(* PLC project Generated.project, CODESYS CODESYS V3.5 SP19 Patch 1 *)
(* stored: creationDateTime 2026-11-18T03:01:31.743540, modificationDateTime 2026-11-18T03:01:31.743540 *)

(* ======================================================================= 💾 ST_Encoder_Calib — Calibration & référence codeur (1 par treuil, RETAIN) ─────────────────────────────────────────────────────────────── 🎯 Rôle : Structure de calibration RETAIN par treuil (M1_EncoderCalib / M2_EncoderCalib) 💾 Données : Références brutes, état homed et contrôle de cohérence redémarrage 📄 Doc métier : DOC/AF/AF_Partie-09_Fonction_Encoder_v2.4.md ======================================================================= *)
TYPE ST_Encoder_Calib : STRUCT
  HomingRefRaw : UDINT;  (* === DONNEES DE REFERENCE BRUTE (RETAIN) === Valeur brute figee au dernier homing reussi *)
  LastKnownRawPos : UDINT;  (* Dernier point brut valide connu (continu) *)
  RestartCoherenceTolerancePts : UDINT := 1000;  (* === CONFIGURATION & REGLAGES TOLERANCE === Tolerance redemarrage (pts, ~12% de 8192) *)
  Homed : BOOL;  (* === ETATS DE CALIBRATION & SECURITE === TRUE des qu'un referencement a reussi *)
  HomingSuspect : BOOL;  (* TRUE si incoherence detectee au redemarrage *)
  HomingProvisional : BOOL;  (* TRUE si zero provisoire 0m HX1 (avant HX4 8.5m) *)
END_STRUCT;
END_TYPE

(* ======================================================================= 🧩 ST_Fault — Brique socle défaut (2 vues : live + latchée) ─────────────────────────────────────────────────────────────── 🎯 Rôle : porter l'état défaut d'un composant, applicable dans TOUS les cas (acquittable ou non), sans brique warning séparée. • Vue LIVE (Error / ErrorId) : suit la cause, retombe seule à 0. • Vue LATCHÉE (Latched / LatchedId): mémorisée au défaut, reste jusqu'au front Reset. Le choix acquittable / non-acquittable se fait PAR CAUSE (ST_FaultCause.Latching), jamais par bloc. 🔒 Sécurité : interlock TOUJOURS sur la cause brute (Error / ErrorId), jamais sur l'acquittement. Reset TOUJOURS effectif, jamais conditionné (std §9). 🧬 Composition : brique de base réutilisable — sortie de FB, struct métier, GVL. Texte IHM NON stocké ici : dérivé côté IHM depuis LatchedId / ErrorId. 📄 Doc : DOC/STDS/CODE_QUALITY_STANDARDS.md §2quinquies / §9 ======================================================================= *)
TYPE ST_Fault : STRUCT
  Error : BOOL;  (* <-- [DIAG] vue LIVE : au moins une cause présente maintenant *)
  ErrorId : WORD;  (* <-- [DIAG] bitfield des causes présentes maintenant (0 si aucune) *)
  Latched : BOOL;  (* <-- [DIAG] vue LATCHÉE : défaut non acquitté, reste jusqu'au front Reset *)
  LatchedId : WORD;  (* <-- [DIAG] ErrorId figé à l'apparition du défaut, effacé au Reset *)
END_STRUCT;
END_TYPE

(* ======================================================================= 🧩 ST_FaultCause — Cause élémentaire alimentant ST_Fault (socle FB_FaultCore) ─────────────────────────────────────────────────────────────── 🎯 Rôle : une cause exprimée EN CLAIR (BOOL + libellé), sans bitfield ni masque. Le FB métier remplit une liste (ARRAY[0..15] OF ST_FaultCause) ; le socle FB_FaultCore en déduit ST_Fault (vue live + vue latchée). 🔒 Sécurité : interlock TOUJOURS sur Active (cause brute), jamais sur le latch. Latching = TRUE → la cause ARME la vue latchée (défaut à acquitter). Latching = FALSE → la cause n'alimente que la vue live (retombe seule). Fail-safe : une cause laissée à Latching=FALSE reste visible en live — pour la rendre acquittable, il faut le déclarer explicitement. 📄 Doc : DOC/STDS/CODE_QUALITY_STANDARDS.md §2quinquies / §9 ======================================================================= *)
TYPE ST_FaultCause : STRUCT
  Active : BOOL;  (* 1 = cause présente maintenant (interlock sur cette valeur) *)
  Latching : BOOL;  (* 1 = cause à acquitter (arme Latched) ; 0 = live seulement *)
  Texte : STRING;  (* libellé prêt IHM (non stocké dans ST_Fault, dérivé côté IHM) *)
END_STRUCT;
END_TYPE

(* ======================================================================= ⚙️ ST_fbEncoder_Cfg — Réglages technologiques publics de FB_Encoder ─────────────────────────────────────────────────────────────────────── 🎯 Rôle : porter le mode de confirmation preset commun aux codeurs. 🔒 Ownership : GVL_IHM.Commun.EncoderCfg ↔ GVL_PERSISTENT._EncoderCfgPersist. 📄 Doc : DOC/AF/AF_Partie-09_Fonction_Encoder_v2.4.md ======================================================================= *)
TYPE ST_fbEncoder_Cfg : STRUCT
  PresetConfirmMode : E_PresetConfirmMode := E_PresetConfirmMode.READBACK_ONLY;  (* Mode de confirmation preset, défaut relecture *)
  Initialized : BOOL := FALSE;  (* 🚦 TRUE après restauration du pont persistant *)
END_STRUCT;
END_TYPE

(* ======================================================================= 🔌 ST_fbEncoder_HwIn — Faits hardware d'entrée codeur (HwIn) ─────────────────────────────────────────────────────────────── 🎯 Rôle : Regrouper les SEULES entrées/faits hardware d'un codeur absolu EtherCAT consommés par FB_Encoder (lecture seule côté automate). 🔒 Ownership : PRG_02_Acquisition câble ce bus depuis le device/simulé. 🛡️ PresetStatusBit : bit du mot d'état codeur, réservé site futur — câblé à FALSE tant qu'aucun bit n'est identifié (aucun signal absent ne confirme implicitement le preset). 📄 Doc métier : DOC/AF/AF_Partie-09_Fonction_Encoder_v2.4.md ======================================================================= *)
TYPE ST_fbEncoder_HwIn : STRUCT
  RawPosIn : UDINT;  (* === ENTRÉES BUS ETHERCAT (faits d'entrée, lecture seule) === --> [HW] Position brute codeur *)
  SpdValueIn : DINT;  (* --> [HW] Vitesse brute codeur (0x6031:01 en 0.1 RPM) *)
  AlarmsIn : UINT;  (* --> [HW] Alarmes brutes codeur *)
  WarningsIn : UINT;  (* --> [HW] Avertissements bruts codeur *)
  SlaveOperational : BOOL;  (* --> [HW] Esclave EtherCAT operationnel *)
  PresetStatusBit : BOOL;  (* --> [HW] Bit d'etat preset optionnel, FALSE si non cable *)
END_STRUCT;
END_TYPE

(* ======================================================================= 🔌 ST_fbEncoder_HwOut — Ordres preset de sortie codeur (HwOut) ─────────────────────────────────────────────────────────────── 🎯 Rôle : Regrouper les SEULES sorties/ordres preset d'un codeur absolu EtherCAT produits par FB_Encoder vers le PDO Rx (bus sortie). 🔒 Ownership : FB_Encoder produit ce bus ; PRG_02_Acquisition le relaie vers le device. 📄 Doc métier : DOC/AF/AF_Partie-09_Fonction_Encoder_v2.4.md ======================================================================= *)
TYPE ST_fbEncoder_HwOut : STRUCT
  PresetTriggerCmd : WORD;  (* === SORTIES BUS ETHERCAT (ordres preset vers PDO Rx) === <-- [ACT] Declenchement preset vers PDO Rx *)
  CodeSeqTriggerCmd : WORD;  (* <-- [ACT] Sequence code vers PDO Rx, maintenue a 0 *)
  PresetValueOut : UDINT;  (* <-- [ACT] Valeur brute envoyee au preset *)
END_STRUCT;
END_TYPE

(* ======================================================================= 📊 ST_fbEncoder_Measurement — Mesures codeur conditionnées (1 sous-DUT par treuil) ─────────────────────────────────────────────────────────────── 🎯 Rôle : Regroupement des mesures et faits de la chaîne codeur d'un treuil (Abs → Scale → Safety → Speed) 🔌 Interface : Interface de mesure normalisée pour PRG_02_Acquisition 📄 Doc métier : DOC/AF/AF_Partie-06_Acquisition_Qualification_IO_v2.4.md ======================================================================= *)
TYPE ST_fbEncoder_Measurement : STRUCT
  RawPos : UDINT;  (* === DONNEES BRUTES & STATUT BUS === Position brute codeur (gelee si EncoderAvailable=FALSE) *)
  EncoderAvailable : BOOL;  (* TRUE = bus/esclave EtherCAT operationnel et disponible *)
  CablePosM : REAL;  (* === MESURES DE POSITION CABLE === Position cable (m, signee, + enroule) *)
  CablePosMSafe : REAL;  (* Position cable instantanee validee par EncoderIncoherent (m) *)
  EncoderIncoherent : BOOL;  (* TRUE = incoherence redemarrage ou hors bornes *)
  Speed_Mps : REAL;  (* === MESURES DE VITESSE CABLE === Vitesse absolue câble (m/s) *)
  SignedSpeed_Mps : REAL;  (* Vitesse signee câble (m/s, + montee, - descente) *)
  SpeedValid : BOOL;  (* TRUE si mesure valide et codeur operationnel *)
  HomingFault : ST_Fault;  (* === STATUTS DES SOUS-FB & REFERENCE === Défaut FB_Encoder_Homing (état du référencement) *)
  HomingLifecycle : ST_Lifecycle;  (* Cycle FB_Encoder_Homing (Busy/Done) *)
  AbsFault : ST_Fault;  (* Défaut FB_Encoder_Abs (état acquisition bus) *)
  HomingRefRaw : UDINT;  (* Reference brute du dernier homing reussi (re-expose) *)
END_STRUCT;
END_TYPE

(* ======================================================================= 🧩 ST_Lifecycle — Brique socle cycle d'exécution ─────────────────────────────────────────────────────────────── 🎯 Rôle : porter l'avancement d'une action à cycle (organe, séquenceur). Optionnelle : un FB purement synchrone (conditionneur, filtre, joystick) ne la porte pas. 🧬 Composition : brique de base réutilisable, composée avec ST_Fault. 📄 Doc : DOC/STDS/CODE_QUALITY_STANDARDS.md §2quinquies ======================================================================= *)
TYPE ST_Lifecycle : STRUCT
  Busy : BOOL;  (* <-- [STAT] 1 = action en cours *)
  Done : BOOL;  (* <-- [STAT] 1 = action terminée avec succès *)
END_STRUCT;
END_TYPE

(* values of E_PresetConfirmMode: READBACK_ONLY: Confirmation par relecture de position; READBACK_AND_STATUSBIT: Relecture et bit d'état matériel; STATUSBIT_ONLY: Bit d'état matériel uniquement *)

{attribute 'qualified_only'}
{attribute 'strict'}
TYPE E_PresetConfirmMode : (READBACK_ONLY := 0, READBACK_AND_STATUSBIT := 1, STATUSBIT_ONLY := 2);
END_TYPE

(* ======================================================================= 🔌 FB_Encoder — Objet codeur complet (1 par treuil M1/M2) ─────────────────────────────────────────────────────────────── 🎯 Rôle : Regrouper toute la chaine codeur derriere une interface unique : Abs → Homing → Scale → Safety → Reliability → Speed. 🔌 Frontiere hardware separee HwIn/HwOut (testable). 🔒 Homing : autorise par HomingPermit (calcule par le caller), declenche par HomingAtTargetM (front). La cible est fournie par le caller. 🔒 Fiabilite : gate EncoderFault (sans Homed) calcule AVANT Speed — purge de vitesse au meme scan. HomedAndReliable = gate strict interlock M3. 🧩 Defaut : Fault:ST_Fault rempli par FB_FaultCore (instFault) depuis une liste de causes en clair (instCauses) — pattern FB_Joystick. Ready = Enable ET pas de defaut late. Interlocks machine sur les faits bruts, jamais sur Fault.Latched. 📄 Doc : DOC/AF/AF_Partie-09_Fonction_Encoder_v2.4.md ======================================================================= *)
FUNCTION_BLOCK FB_Encoder
  VAR_INPUT
    Enable : BOOL;  (* === COMMANDES & AUTORISATIONS === --> [CMD] Autorisation generale FB (TRUE=Autorise) *)
    Reset : BOOL;  (* --> [CMD] Acquittement defaut (front montant) *)
    HomingPermit : BOOL;  (* === AUTORISATION HOMING (calculee par le caller PRG) === --> [CMD] TRUE = l'operateur a le droit de homer *)
    HomingAtTargetM : BOOL;  (* === CONSIGNES HOMING === --> [CMD] Demande homing vers cible (front montant) *)
    HomingAtZero : BOOL;  (* --> [CMD] Force homing a 0.0 *)
    ConfirmCoherence : BOOL;  (* --> [CMD] Lever le doute d'incoherence boot *)
    CfgHomingTargetM : REAL;  (* --> [CFG] Cible libre homing unitaire (m) *)
    CfgTopSensorPosM : REAL;  (* --> [CFG] Cible homing nominal capteur haut (m) *)
    UseDynamicTarget : BOOL;  (* --> [CMD] Active cible dynamique *)
    DynamicHomingTargetM : REAL;  (* --> [CFG] Cible dynamique de referencement (m) *)
    InvalidateDatum : BOOL := FALSE;  (* --> [CMD] Invalidation explicite du datum (abandon homing avant altimetrie) *)
    ProvisionalHoming : BOOL := FALSE;  (* --> [CMD] TRUE = zero provisoire HX1 (survive coupure secteur RETAIN) *)
    TopPositionSensor : BOOL;  (* === CAPTEURS PHYSIQUES === --> [HW] Capteur physique position haute unique *)
    HwIn : ST_fbEncoder_HwIn;  (* === BUS ETHERCAT & CAPTEUR HW (frontiere testable) === --> [HW] Retours hardware codeur *)
    PointsPerRev : UDINT := 8192;  (* === MECANIQUE (constantes) === --> [CFG] Resolution codeur (pts/tour) *)
    CableM_PerRev : REAL := 2;  (* --> [CFG] Developpement cable par tour (m/tour) *)
    Cfg : ST_fbEncoder_Cfg;  (* === REGLAGES & CONFIGURATION === --> [CFG] Mode de confirmation preset *)
    PositionMinM : REAL := -99;  (* --> [CFG] Plafond bornage physique bas (m) *)
    PositionMaxM : REAL := 99;  (* --> [CFG] Plafond bornage physique haut (m) *)
    BypassGlobal : BOOL := FALSE;  (* --> [TST] Neutralisation defauts pour mise en service *)
  END_VAR
  VAR_OUTPUT
    Ready : BOOL;  (* === ETATS IEC & SYNOPTIQUE === <-- [STAT] FB pret a fonctionner (Enable ET pas de defaut late) *)
    Fault : ST_Fault;  (* <-- [DIAG] Brique defaut socle (live + latchee), remplie par FB_FaultCore *)
    HwOut : ST_fbEncoder_HwOut;  (* === FRONTIERE HW SORTIE (testable) === <-- [ACT] Ordres hardware codeur (preset) *)
    Measurement : ST_fbEncoder_Measurement;  (* === MESURES CONDITIONNEES (struct frontiere) === <-- [BUS] Mesures + statuts (interface) *)
    Homed : BOOL;  (* === ETATS CODEUR === <-- [STAT] Codeur reference (sortie homing) *)
    HomingSuspect : BOOL;  (* <-- [DIAG] Incoherence redemarrage a lever *)
    HomingProvisional : BOOL;  (* <-- [STAT] TRUE si datum provisoire RETAIN actif (HX1 0m) *)
    EncoderFault : BOOL;  (* <-- [SAFE] Gate general fiabilite (sans Homed) *)
    HomedAndReliable : BOOL;  (* <-- [STAT] Gate strict M3 : dispo ET ref ET pas incoherent *)
    PresetConfirmationFailed : BOOL;  (* <-- [DIAG] Latch derniere verification preset echouee *)
  END_VAR
  VAR_IN_OUT
    Calib : ST_Encoder_Calib;  (* === CALIBRATION PERSISTANTE (externe RETAIN, jamais membre) === <-> [BUS] Calibration RETAIN du treuil *)
  END_VAR
  VAR
    instAbs : FB_Encoder_Abs;  (* === SOUS-INSTANCES FB (chaine codeur complete) === * [INST] Acquisition brute codeur EtherCAT *)
    instHoming : FB_Encoder_Homing;  (* * [INST] Referencement (homing) nominal/unitaire *)
    instScale : FB_Encoder_Scale;  (* * [INST] Mise a l'echelle points -> metres *)
    instSafety : FB_Encoder_Safety;  (* * [INST] Bornage & coherence mesure *)
    instRel : FB_EncoderReliability;  (* * [INST] Gates de fiabilite *)
    instSpeed : FB_Encoder_SpeedMeasure;  (* * [INST] Calcul vitesse cable *)
    instFault : FB_FaultCore;  (* * [INST] Socle de defaut (liste de causes -> ST_Fault) *)
    instCauses : ARRAY[0..15] OF ST_FaultCause;  (* . [LOC] Liste des causes pour le socle FB_FaultCore *)
  END_VAR

            

{region "§1 Gate neutralisation"}
IF NOT Enable THEN
    Ready := FALSE;
    Measurement.RawPos := 0; Measurement.EncoderAvailable := FALSE;
    Measurement.CablePosM := 0.0; Measurement.CablePosMSafe := 0.0; Measurement.EncoderIncoherent := FALSE;
    Measurement.Speed_Mps := 0.0; Measurement.SignedSpeed_Mps := 0.0; Measurement.SpeedValid := FALSE;
    Measurement.HomingFault.Error := FALSE; Measurement.HomingFault.ErrorId := 0;
    Measurement.HomingLifecycle.Busy := FALSE; Measurement.HomingLifecycle.Done := FALSE;
    Measurement.AbsFault.Error := FALSE;    Measurement.AbsFault.ErrorId := 0;
    EncoderFault := TRUE;
    HomedAndReliable := FALSE;
    // Frontiere HW sortie : aucun ordre preset publie hors autorisation
    // (sinon PRG_02_Acquisition relaie une valeur perimee au codeur absolu -> preset parasite, reference corrompue)
    HwOut.PresetTriggerCmd := 0; HwOut.CodeSeqTriggerCmd := 0; HwOut.PresetValueOut := 0;
    // Reference connue MAINTENUE depuis Calib (RETAIN) meme FB desactive (AF09 §4) :
    // un FB desactive ne doit pas faire perdre la reference aux consommateurs aval (PRG_04, FB_Encoder_Scale).
    Homed := Calib.Homed;
    HomingSuspect := Calib.HomingSuspect;
    HomingProvisional := Calib.HomingProvisional;
    Measurement.HomingRefRaw := Calib.HomingRefRaw;
    // PresetConfirmationFailed est un diagnostic latch : il reste gele hors Enable
    // et ne doit pas etre efface par ce gate (AC3).
    // Socle appele meme Enable=FALSE : maintient le latch non acquitte et traite le Reset
    // hors autorisation (AC4). Les causes ne sont pas evaluees (Enable=FALSE -> vue live a 0),
    // les latches sont preserves.
    instFault(Enable := FALSE, Reset := Reset, Causes := instCauses);
    Fault := instFault.Fault;
    RETURN;
END_IF;
Ready := TRUE;
{endregion}

{region "§2 Abs"}
    instAbs(
    Enable              := Enable,
    Reset               := Reset,
    RawPosIn            := HwIn.RawPosIn,
    AlarmsIn            := HwIn.AlarmsIn,
    WarningsIn          := HwIn.WarningsIn,
    SlaveOperational    := HwIn.SlaveOperational,
    PresetRequest       := instHoming.PresetRequest,
    PresetValue         := instHoming.PresetValue,
    PointsPerRev        := PointsPerRev
);
{endregion}

{region "§3 Homing"}
instHoming(
    Enable               := Enable,
    Reset                := Reset,
    Home                 := HomingAtTargetM,
    HomingPermit         := HomingPermit,
    BtnConfirmCoherence  := ConfirmCoherence,
    InvalidateDatum      := InvalidateDatum,
    ProvisionalHoming    := ProvisionalHoming,
    UseDynamicTarget     := UseDynamicTarget,
    DynamicHomingTargetM := DynamicHomingTargetM,
    CfgHomingTargetM     := CfgHomingTargetM,
    CfgTopSensorPosM     := SEL(HomingAtZero, CfgTopSensorPosM, 0.0),
    TopPositionSensor    := TopPositionSensor,
    RawPos               := instAbs.RawPos,
    EncoderAvailable     := instAbs.EncoderAvailable,
    PresetStatusBit      := HwIn.PresetStatusBit,
    Cfg                  := Cfg,
    PointsPerRev         := PointsPerRev,
    MultiTurnRevsMax     := 4096,
    CableM_PerRev        := CableM_PerRev,
    BypassGlobal         := BypassGlobal,
    Calib                := Calib
);
{endregion}

{region "§4 Scale"}
instScale(
    RawPos       := instAbs.RawPos,
    HomingRefRaw := instHoming.HomingRefRaw,
    CableM_PerRev := CableM_PerRev,
    PointsPerRev := PointsPerRev
);
{endregion}

{region "§5 Safety"}
instSafety(
    Enable             := Enable,
    Reset              := Reset,
    CablePosM          := instScale.CablePosM,
    HomingSuspect      := instHoming.HomingSuspect,
    PositionMinM       := PositionMinM,
    PositionMaxM       := PositionMaxM,
    BypassGlobal       := BypassGlobal
);
{endregion}

{region "§6 Reliability"}
instRel(
    EncoderAvailable  := instAbs.EncoderAvailable,
    Homed             := instHoming.Homed,
    EncoderIncoherent := instSafety.EncoderIncoherent
);
{endregion}

{region "§7 Speed"}
instSpeed(
    Enable        := Enable,
    Reset         := Reset,
    SpdValueIn    := HwIn.SpdValueIn,
    PositionValid := NOT instRel.EncoderFault,
    CableM_PerRev := CableM_PerRev
);
{endregion}

{region "§8 Remplissage struct et synthese"}
Measurement.RawPos            := instAbs.RawPos;
Measurement.EncoderAvailable  := instAbs.EncoderAvailable;
Measurement.CablePosM         := instSafety.CablePosMSafe;
Measurement.CablePosMSafe     := instSafety.CablePosMSafe;
Measurement.EncoderIncoherent := instSafety.EncoderIncoherent;
Measurement.Speed_Mps         := instSpeed.Speed_Mps;
Measurement.SignedSpeed_Mps   := instSpeed.SignedSpeed_Mps;
Measurement.SpeedValid        := instSpeed.Valid;
Measurement.HomingFault        := instHoming.Fault;
Measurement.HomingLifecycle    := instHoming.Lifecycle;
Measurement.AbsFault           := instAbs.Fault;
Measurement.HomingRefRaw      := instHoming.HomingRefRaw;

// Frontiere HW sortie (preset)
HwOut.PresetTriggerCmd := instAbs.PresetTriggerCmd;
HwOut.CodeSeqTriggerCmd := instAbs.CodeSeqTriggerCmd;
HwOut.PresetValueOut    := instAbs.PresetValueOut;

// Etats codeur
Homed            := instHoming.Homed;
HomingSuspect    := instHoming.HomingSuspect;
HomingProvisional := instHoming.HomingProvisional;
EncoderFault     := instRel.EncoderFault;
HomedAndReliable := instRel.HomedAndReliable;
PresetConfirmationFailed := instHoming.PresetConfirmationFailed;

// Synthese statut facade : brique defaut socle (Fault:ST_Fault), pattern FB_Joystick.
// Causes exprimees en CLAIR (ST_FaultCause), alimentees UNIQUEMENT depuis les sorties
// publiques des sous-FB (encapsulation stricte, jamais de lecture VAR interne).
//   - Cause 0/1 : LIVE (Latching=FALSE) -> Fault.Error, retombe seule.
//   - Cause 2   : LATCHED (Latching=TRUE) -> arme Fault.Latched, acquittee au Reset front.
// Interlock machine toujours sur les faits bruts (EncoderFault, HomedAndReliable,
// EncoderIncoherent), jamais sur Fault.Latched (conservation).
instCauses[0].Active := NOT instAbs.EncoderAvailable; instCauses[0].Latching := FALSE;
instCauses[0].Texte := 'Perte materiel / communication codeur EtherCAT';
instCauses[1].Active := instSafety.EncoderIncoherent; instCauses[1].Latching := FALSE;
instCauses[1].Texte := 'Incoherence mesure / saut de position codeur';
instCauses[2].Active := instHoming.PresetConfirmationFailed; instCauses[2].Latching := TRUE;
instCauses[2].Texte := 'Echec confirmation transaction preset codeur';

// Socle appele APRES le pipeline : causes du scan courant, aucun scan de retard (AC4).
instFault(Enable := Enable, Reset := Reset, Causes := instCauses);
Fault := instFault.Fault;     // source de verite = socle
Ready := Enable AND NOT Fault.Latched;
{endregion}

          
END_FUNCTION_BLOCK

(* ======================================================================= 🛡️ FB_EncoderReliability — Gates de fiabilite de la chaine codeur ─────────────────────────────────────────────────────────────── 🎯 Rôle : Synthetise les gates de fiabilite d'un treuil a partir des faits produits par la chaine codeur (Abs/Homing/Safety), pur calcul combinatoire, sans memoire ni machine d'etat. 🔒 Polarité : EncoderFault = NOT EncoderAvailable OR EncoderIncoherent (gate GENERAL, SANS Homed) HomedAndReliable = EncoderAvailable AND Homed AND NOT EncoderIncoherent (gate STRICT M3) 🧩 Responsabilite scindee (D-A2bis) : Homing = referencement, Safety = coherence, ce FB = « le codeur est fiable ». Aucune recomposition chez les consommateurs. 📄 Doc : DOC/AF/AF_Partie-09_Fonction_Encoder_v2.4.md ======================================================================= *)
FUNCTION_BLOCK FB_EncoderReliability
  VAR_INPUT
    EncoderAvailable : BOOL;  (* === FAITS DE LA CHAINE CODEUR === --> [HW] Codeur operationnel sur bus (FB_Encoder_Abs) *)
    Homed : BOOL;  (* --> [STAT] Codeur reference (FB_Encoder_Homing) *)
    EncoderIncoherent : BOOL;  (* --> [SAFE] Incoherence ou hors bornes (FB_Encoder_Safety) *)
  END_VAR
  VAR_OUTPUT
    EncoderFault : BOOL;  (* === GATES DE FIABILITE === <-- [SAFE] Gate general fiabilite (SANS Homed) — vitesse/mouvements *)
    HomedAndReliable : BOOL;  (* <-- [STAT] Gate strict M3 : disponible ET reference ET pas incoherent *)
  END_VAR

            

// 🛡️ 1. GATE GENERAL (D-A11, C1) — PAS de Homed : non-reference ≠ incoherent.
//    Ce gate sert a la fiabilite de la mesure (vitesse, mouvements, PositionsValid).
EncoderFault := (NOT EncoderAvailable) OR EncoderIncoherent;

// 🎯 2. GATE STRICT — reserve a l'interlock hauteur M3 (C1) : on ne translate pas
//    si la hauteur est inconnue (jamais home) ou douteuse.
HomedAndReliable := EncoderAvailable AND Homed AND (NOT EncoderIncoherent);

          
END_FUNCTION_BLOCK

(* ======================================================================= 🔌 FB_Encoder_Abs — Acquisition codeur absolu (accès bus EtherCAT) ─────────────────────────────────────────────────────────────── 🎯 Rôle : Accès bus EtherCAT, extraction positions brutes et séquence de Preset SDO 🔒 Polarité : EncoderAvailable=TRUE si communication bus et esclave OK 🔌 Architecture : Module d'acquisition codeur absolu 📄 Doc métier : DOC/AF/AF_Partie-09_Fonction_Encoder_v2.4.md ======================================================================= === DECLARATION (à coller dans la partie déclaration du POU FB_Encoder_Abs) === *)
FUNCTION_BLOCK FB_Encoder_Abs
  VAR_INPUT
    Enable : BOOL;  (* === COMMANDES & AUTORISATIONS === --> [CMD] Autorisation generale FB (TRUE=Autorise) *)
    Reset : BOOL;  (* --> [CMD] Acquittement defaut (front montant) *)
    PresetRequest : BOOL;  (* --> [CMD] Demande de preset (front montant) *)
    RawPosIn : UDINT;  (* === BUS ETHERCAT & CAPTEUR HW === --> [HW] Position brute EtherCAT *)
    AlarmsIn : UINT;  (* --> [HW] Codes alarmes bruts EtherCAT *)
    WarningsIn : UINT;  (* --> [HW] Codes avertissements bruts EtherCAT *)
    SlaveOperational : BOOL;  (* --> [HW] Statut esclave EtherCAT operationnel *)
    PointsPerRev : UDINT := 8192;  (* === PARAMETRES & REGLAGES === --> [CFG] Resolution codeur (pts/tour) *)
    PresetValue : UDINT;  (* --> [CFG] Valeur cible de preset *)
    PresetTimeout : TIME := TIME#2s0ms;  (* --> [CFG] Temporisation max attente preset *)
    PresetTolerancePts : UDINT := 10;  (* --> [CFG] Tolerance relecture post-preset (pts) *)
  END_VAR
  VAR_OUTPUT
    Ready : BOOL;  (* === ETATS IEC & SYNOPTIQUE === <-- [STAT] FB pret a fonctionner *)
    Fault : ST_Fault;  (* 🧩 Statut transverse (forme cible ST_Fault) *)
    RawPos : UDINT;  (* === MESURES & DONNEES CODEUR === <-- [DIAG] Position brute gelee si non disponible *)
    EncoderAvailable : BOOL;  (* <-- [STAT] Codeur operationnel et disponible *)
    AngleRaw : UINT;  (* <-- [DIAG] Angle brut sur un tour (MOD PointsPerRev) *)
    TurnCount : UDINT;  (* <-- [DIAG] Nombre de tours bruts (RawPos / PointsPerRev) *)
    PresetTriggerCmd : WORD;  (* === COMMANDES & ECHANGE BUS ETHERCAT === <-- [ACT] Ordre declenchement preset vers PDO Rx *)
    CodeSeqTriggerCmd : WORD;  (* <-- [ACT] Ordre sequence code vers PDO Rx *)
    PresetValueOut : UDINT;  (* <-- [ACT] Valeur de preset transmise au PDO Rx *)
  END_VAR
  VAR
    ResetEdge : R_TRIG;  (* === DETECTEURS DE FRONT === . [LOC] Detecteur front montant Reset *)
    PresetReqEdge : R_TRIG;  (* . [LOC] Detecteur front montant PresetRequest *)
    PresetTimer : TON;  (* === TEMPORISATEURS INTERNES === . [LOC] Temporisateur timeout sequence preset *)
    PresetTimerVisual : TON;  (* . [LOC] Temporisateur maintien visuel impulsion (500ms) *)
    PresetSeqStep : INT;  (* === VARIABLES INTERNES DE CALCUL & ETAT === . [LOC] Etape sequence preset (0:IDLE, 1:PULSE/WAIT) *)
    RawDiff : DINT;  (* . [LOC] Ecart signe entre RawPos et PresetValueOut *)
    PresetCompleted : BOOL;  (* . [LOC] Fait de fin de maintien preset (un scan) *)
    PresetTimeoutError : BOOL;  (* . [LOC] Latch interne timeout séquence preset *)
    instFault : FB_FaultCore;  (* === SOCLE DEFAUT (FB_FaultCore) === * [INST] Socle défaut transverse *)
    instCauses : ARRAY[0..15] OF ST_FaultCause;  (* . [LOC] Table des causes nommées *)
  END_VAR

            

// === IMPLEMENTATION (à coller dans le corps ST du POU FB_Encoder_Abs) ===

{region "§1 Causes & Socle Défaut (évalué en continu)"}
// 🔑 1. RESET FRONT
ResetEdge(CLK := Reset);

// 🔍 2. DIAGNOSTIC BUS / ALARME (Cause 0 : live)
instCauses[0].Active   := (AlarmsIn <> 0) OR NOT SlaveOperational;
instCauses[0].Latching := FALSE;
instCauses[0].Texte    := 'Defaut communication EtherCAT codeur absolu';

// ⏱️ 3. TIMEOUT PRESET (Cause 1 : latched)
IF ResetEdge.Q AND (PresetSeqStep = 0) THEN
    PresetTimeoutError := FALSE;
END_IF;
instCauses[1].Active   := PresetTimeoutError;
instCauses[1].Latching := TRUE;
instCauses[1].Texte    := 'Timeout sequence preset SDO codeur';

// Appel du socle de défaut
instFault(Enable := Enable, Reset := Reset, Causes := instCauses);
Fault := instFault.Fault;

EncoderAvailable := NOT instCauses[0].Active;
{endregion}

{region "§2 Gate neutralisation"}
// 🛑 2. GATE
IF NOT Enable THEN
    EncoderAvailable := FALSE;
    Ready := FALSE;
    PresetTriggerCmd := 0; CodeSeqTriggerCmd := 0; PresetValueOut := 0;
    PresetSeqStep := 0;
    PresetCompleted := FALSE;
    PresetTimer(IN := FALSE, PT := PresetTimeout);
    PresetTimerVisual(IN := FALSE, PT := T#500MS);
    // RawPos, AngleRaw et TurnCount sont volontairement gelés hors Enable
    // (AF09 F09.01 / AC5) : aucune lecture bus ni remise a zero dans ce gate.
    RETURN;
END_IF;

Ready := Enable AND NOT Fault.Latched;
{endregion}

{region "§3 Lecture position"}
// 📥 3. LECTURE POSITION — GELER SUR DOUTE (Partie10 §6)
// Si EncoderAvailable=FALSE : RawPos/AngleRaw/TurnCount conservent leur dernière valeur (pas de RETURN
// global ici pour ne pas geler aussi la séquence preset/l'état — seule la lecture est gelée).
IF EncoderAvailable THEN
    RawPos := RawPosIn;   // Sens de comptage géré côté codeur (CoE 6000h bit0, startup parameter CODESYS) — voir Partie10 §3bis. Plus de calcul ici.
    AngleRaw := UDINT_TO_UINT(RawPos MOD PointsPerRev);
    TurnCount := RawPos / PointsPerRev;
END_IF;
{endregion}

{region "§4 Séquence preset"}
// 🔧 4. SÉQUENCE PRESET (écriture bus)
// PresetTriggerCmd := 2 déclenche le référencement à PresetValue (valeur de commande, pas un
// masque de bits). CodeSeqTriggerCmd : rôle non identifié — laissé à 0, PAS piloté tant que sa
// fonction n'est pas confirmée. Ne jamais lui donner une valeur arbitraire.
PresetReqEdge(CLK := PresetRequest);
PresetCompleted := FALSE;
CodeSeqTriggerCmd := 0;                 // non piloté — rôle inconnu, voir note ci-dessus
CASE PresetSeqStep OF
    0: // IDLE
        PresetTriggerCmd := 0;
        IF PresetReqEdge.Q AND EncoderAvailable THEN
            PresetValueOut := PresetValue;
            PresetSeqStep := 1;
            PresetTimer(IN := TRUE, PT := PresetTimeout);
        END_IF;
    1: // Déclenchement preset (laissé actif pendant 0.5s pour confort visuel en simulation/bus)
        PresetTriggerCmd := 2;   // Référence le codeur à PresetValueOut
        RawDiff := UDINT_TO_DINT(RawPos) - UDINT_TO_DINT(PresetValueOut);
        IF ABS(RawDiff) <= UDINT_TO_DINT(PresetTolerancePts) THEN
            PresetTimer(IN := FALSE, PT := PresetTimeout);
            PresetTimerVisual(IN := TRUE, PT := T#500MS);
            IF PresetTimerVisual.Q THEN
                PresetTriggerCmd := 0;
                PresetCompleted := TRUE;
                PresetSeqStep := 0;
                PresetTimerVisual(IN := FALSE, PT := T#500MS);
            END_IF;
        ELSIF PresetTimer.Q THEN
            PresetTriggerCmd := 0;
            PresetTimeoutError := TRUE;
            PresetSeqStep := 0;
            PresetTimer(IN := FALSE, PT := PresetTimeout);
            PresetTimerVisual(IN := FALSE, PT := T#500MS);
        END_IF;
END_CASE;
{endregion}

          
END_FUNCTION_BLOCK

(* ======================================================================= ⚙️ FB_Encoder_Homing — Référencement codeur nominal ou unitaire ─────────────────────────────────────────────────────────────── 🎯 Rôle : Séquence de référencement nominal (capteur haut) ou unitaire (MAINT_N2) 🔒 Polarité : Homed=TRUE dès qu'un référencement valide est enregistré 🔌 Architecture : Expose ST_Encoder_Calib en VAR_IN_OUT 📄 Doc métier : DOC/AF/AF_Partie-09_Fonction_Encoder_v2.4.md ======================================================================= === DECLARATION (à coller dans la partie déclaration du POU FB_Encoder_Homing) === *)
FUNCTION_BLOCK FB_Encoder_Homing
  VAR_INPUT
    Enable : BOOL;  (* === COMMANDES & AUTORISATIONS === --> [CMD] Autorisation generale FB (TRUE=Autorise) *)
    Reset : BOOL;  (* --> [CMD] Acquittement defaut (front montant) *)
    Home : BOOL;  (* --> [CMD] Demande de referencement (front) *)
    HomingPermit : BOOL;  (* --> [CMD] Autorisation de homer (calculee par le caller) *)
    BtnConfirmCoherence : BOOL;  (* --> [CMD] Levee de doute d'incoherence au boot (front) *)
    InvalidateDatum : BOOL := FALSE;  (* --> [CMD] Invalidation explicite du datum (abandon avant calibration finale) *)
    ProvisionalHoming : BOOL := FALSE;  (* --> [CMD] TRUE = preset provisoire (ex. 0m HX1), FALSE = definitif *)
    CfgHomingTargetM : REAL;  (* === CIBLES & CONFIGURATION HOMING === --> [CFG] Cible libre homing unitaire (m) *)
    UseDynamicTarget : BOOL := FALSE;  (* --> [CFG] Activation cible dynamique *)
    DynamicHomingTargetM : REAL := 0;  (* --> [CFG] Cible dynamique de referencement (m) *)
    CfgTopSensorPosM : REAL := 8.5;  (* --> [CFG] Cible homing nominal capteur haut (m) *)
    TopPositionSensor : BOOL;  (* === RETOURS HW & CAPTEURS === --> [HW] Capteur physique position haute unique *)
    RawPos : UDINT;  (* === MESURES & RETOURS FB CODEUR ABSOLU === --> [HW] Position brute codeur (sortie FB_Encoder_Abs) *)
    EncoderAvailable : BOOL;  (* --> [HW] Codeur absolu disponible et valide *)
    PresetStatusBit : BOOL;  (* --> [HW] Bit d'etat preset optionnel, FALSE si non cable *)
    Cfg : ST_fbEncoder_Cfg;  (* === REGLAGES TRANSACTION PRESET === --> [CFG] Mode de confirmation preset *)
    PointsPerRev : UDINT := 8192;  (* === CARACTERISTIQUES MECANIQUES & BUS === --> [CFG] Resolution codeur (pts/tour) *)
    MultiTurnRevsMax : UDINT := 4096;  (* --> [CFG] Capacite multitour max codeur (tours) *)
    CableM_PerRev : REAL := 2;  (* --> [CFG] Perimetre tambour / developpement cable (m/tour) *)
    BypassGlobal : BOOL := FALSE;  (* === TESTS & BYPASS === --> [TST] Neutralisation securites pour mise en service *)
  END_VAR
  VAR_OUTPUT
    Ready : BOOL;  (* === ETATS IEC & SYNOPTIQUE === <-- [STAT] FB pret a fonctionner *)
    Fault : ST_Fault;  (* 🧩 Statut transverse (forme cible ST_Fault) *)
    Lifecycle : ST_Lifecycle;  (* 🧩 Cycle de vie (forme cible ST_Lifecycle) *)
    PresetRequest : BOOL;  (* === COMMANDES VERS FB_ENCODER_ABS === <-- [ACT] Pulse demande d'ecriture preset SDO *)
    PresetValue : UDINT;  (* <-- [ACT] Valeur de cible brute pour preset SDO *)
    Homed : BOOL;  (* === RESULTATS & MEMOIRE CALIBRATION === <-- [STAT] Codeur pagine et referencie *)
    HomingSuspect : BOOL;  (* <-- [DIAG] Incoherence redemarrage a lever *)
    HomingProvisional : BOOL;  (* <-- [STAT] TRUE si datum provisoire RETAIN actif (HX1 0m) *)
    HomingRefRaw : UDINT;  (* <-- [DIAG] Offset de reference brut calcule *)
    PresetConfirmationFailed : BOOL;  (* <-- [DIAG] Latch derniere verification preset echouee *)
  END_VAR
  VAR_IN_OUT
    Calib : ST_Encoder_Calib;  (* === STRUCTURE DE CALIBRATION PERSISTANTE === <-> [BUS] Structure de calibration RETAIN *)
  END_VAR
  VAR
    ResetEdge : R_TRIG;  (* === DETECTEURS DE FRONT === . [LOC] Detecteur front montant Reset *)
    HomeEdge : R_TRIG;  (* . [LOC] Detecteur front montant Home *)
    ConfirmCoherenceEdge : R_TRIG;  (* . [LOC] Detecteur front montant BtnConfirmCoherence *)
    TopSensorEdge : R_TRIG;  (* . [LOC] Detecteur front montant TopPositionSensor *)
    DynamicTargetEdge : R_TRIG;  (* . [LOC] Detecteur front montant UseDynamicTarget *)
    InitDone : BOOL;  (* === ETATS & DRAPEAUX INTERNES === . [LOC] Controle incoherence boot effectue *)
    HomingModeOk : BOOL;  (* . [LOC] Mode de fonctionnement valide pour homing *)
    NominalHomingTrigger : BOOL;  (* . [LOC] Condition de declenchement homing nominal *)
    UnitaryHomingTrigger : BOOL;  (* . [LOC] Condition de declenchement homing unitaire *)
    DynamicHomingTrigger : BOOL;  (* . [LOC] Condition de declenchement homing dynamique *)
    HomingTrigger : BOOL;  (* . [LOC] Synthese declenchement homing *)
    PresetVerificationActive : BOOL;  (* . [LOC] Verification preset en attente *)
    PendingProvisional : BOOL;  (* . [LOC] Capture mode provisoire pendant verification preset *)
    PresetConfirmed : BOOL;  (* . [LOC] Resultat du mode de confirmation selectionne *)
    HomingModeError : BOOL;  (* === DRAPEAUX DEFAUTS INTERNES === . [LOC] Latch erreur mode *)
    TargetOutOfRangeError : BOOL;  (* . [LOC] Latch cible hors limites *)
    PresetFailError : BOOL;  (* . [LOC] Latch échec preset *)
    BootIncoherentError : BOOL;  (* . [LOC] Latch incohérence boot *)
    TargetPoints : DINT;  (* === VARIABLES DE CALCUL === . [LOC] Ecart cible converti en points *)
    TargetPositionM : REAL;  (* . [LOC] Cible retenue en metres *)
    RawDiffRestart : DINT;  (* . [LOC] Ecart brut de position au redemarrage *)
    PendingHomingRefRaw : UDINT;  (* . [LOC] Reference candidate, non publiee avant succes *)
    CandidateRawDiff : DINT;  (* . [LOC] Ecart brut de la mesure candidate *)
    CandidateCablePosM : REAL;  (* . [LOC] Position candidate calculee avant commit *)
    ReadbackOk : BOOL;  (* . [LOC] Mesure candidate dans la tolerance *)
    StatusBitOk : BOOL;  (* . [LOC] Etat du bit optionnel de confirmation *)
    PresetVerifyTimer : TON;  (* . [LOC] Temporisation historique de verification 500ms *)
    instFault : FB_FaultCore;  (* === SOCLE DEFAUT (FB_FaultCore) === * [INST] Socle défaut transverse *)
    instCauses : ARRAY[0..15] OF ST_FaultCause;  (* . [LOC] Table des causes nommées *)
    CST_HomingVerifyToleranceM : REAL := 0.01;  (* === TOLERANCE & TEMPORISATION TRANSACTION === Tolerance mesure cible (m) *)
    CST_PresetVerifyTime : TIME := TIME#50MS;  (* Latence historique avant relecture *)
  END_VAR

            

// === IMPLEMENTATION (à coller dans le corps ST du POU FB_Encoder_Homing) ===

{region "§1 Causes & Socle Défaut (évalué en continu)"}
// 🔑 1. FRONTS
ResetEdge(CLK := Reset);
HomeEdge(CLK := Home);
ConfirmCoherenceEdge(CLK := BtnConfirmCoherence);

// Effacement des latches d'erreur sur Reset conscient
IF ResetEdge.Q THEN
    PresetConfirmationFailed := FALSE;
    HomingModeError := FALSE;
    TargetOutOfRangeError := FALSE;
    PresetFailError := FALSE;
END_IF;

// Levée de doute incohérence boot (BtnConfirmCoherence)
IF ConfirmCoherenceEdge.Q THEN
    Calib.HomingSuspect := FALSE;
    BootIncoherentError := FALSE;
END_IF;

// Configuration des causes nommées
instCauses[0].Active   := HomingModeError;
instCauses[0].Latching := TRUE;
instCauses[0].Texte    := 'Homing non autorise dans ce mode';

instCauses[1].Active   := TargetOutOfRangeError;
instCauses[1].Latching := TRUE;
instCauses[1].Texte    := 'Cible de homing hors plage';

instCauses[2].Active   := PresetFailError;
instCauses[2].Latching := TRUE;
instCauses[2].Texte    := 'Echec confirmation transaction preset';

instCauses[3].Active   := BootIncoherentError;
instCauses[3].Latching := TRUE;
instCauses[3].Texte    := 'Incoherence position codeur au demarrage';

// Appel du socle de défaut
instFault(Enable := Enable, Reset := Reset, Causes := instCauses);
Fault := instFault.Fault;
{endregion}

{region "§2 Gate neutralisation"}
// 🛑 2. GATE — neutralisation ; on continue toutefois d'exposer le dernier état RETAIN connu
// (FB_Encoder_Scale a besoin de HomingRefRaw même si ce FB est désactivé)
IF NOT Enable THEN
    PresetRequest := FALSE;
    PresetValue := 0;
    Ready := FALSE;
    Lifecycle.Busy := FALSE;
    Lifecycle.Done := FALSE;
    InitDone := FALSE;   // Force un nouveau contrôle à la prochaine activation
    PresetVerificationActive := FALSE;
    PresetVerifyTimer(IN := FALSE, PT := CST_PresetVerifyTime);
    Homed := Calib.Homed;
    HomingSuspect := Calib.HomingSuspect;
    HomingProvisional := Calib.HomingProvisional;
    HomingRefRaw := Calib.HomingRefRaw;
    // PresetConfirmationFailed est un diagnostic latch : il est gelé hors Enable
    RETURN;
END_IF;

Ready := Enable AND NOT Fault.Latched;
{endregion}

IF InvalidateDatum THEN
    Calib.Homed              := FALSE;
    Calib.HomingSuspect      := FALSE;
    Calib.HomingProvisional  := FALSE;
    PendingProvisional       := FALSE;
    Lifecycle.Done           := FALSE;
    PresetVerificationActive := FALSE;
    PresetVerifyTimer(IN := FALSE, PT := CST_PresetVerifyTime);
END_IF;

{region "§3 Cohérence au redémarrage"}
// 🔍 3. COHÉRENCE AU REDÉMARRAGE — une fois par session Enable, dès que le codeur répond
IF NOT InitDone THEN
    IF EncoderAvailable THEN
        RawDiffRestart := UDINT_TO_DINT(RawPos) - UDINT_TO_DINT(Calib.LastKnownRawPos);
        IF Calib.Homed AND (ABS(RawDiffRestart) > UDINT_TO_DINT(Calib.RestartCoherenceTolerancePts)) THEN
            Calib.HomingSuspect := TRUE;
            BootIncoherentError := TRUE;
        END_IF;
        InitDone := TRUE;
    END_IF;
END_IF;
{endregion}

{region "§4 Demande et déclenchement homing"}
// ⚙️ 4. DEMANDE & DÉCLENCHEMENT HOMING
PresetRequest := FALSE;
PresetValue := 0;
TopSensorEdge(CLK := TopPositionSensor);
DynamicTargetEdge(CLK := UseDynamicTarget);

HomingModeOk := HomingPermit;

IF HomeEdge.Q AND NOT HomingModeOk THEN
    HomingModeError := TRUE;
END_IF;

NominalHomingTrigger := HomingModeOk AND NOT UseDynamicTarget
                         AND ((Home AND TopSensorEdge.Q) OR (HomeEdge.Q AND TopPositionSensor));

UnitaryHomingTrigger := HomingModeOk AND NOT UseDynamicTarget AND HomeEdge.Q;

DynamicHomingTrigger := HomingModeOk AND (DynamicTargetEdge.Q OR (UseDynamicTarget AND HomeEdge.Q));

HomingTrigger := (NominalHomingTrigger OR UnitaryHomingTrigger OR DynamicHomingTrigger)
                 AND NOT PresetVerificationActive;

IF HomingTrigger THEN
    IF UseDynamicTarget THEN
        TargetPositionM := DynamicHomingTargetM;
    ELSIF NominalHomingTrigger THEN
        TargetPositionM := CfgTopSensorPosM;
    ELSE
        TargetPositionM := CfgHomingTargetM;
    END_IF;

    // Bornage obligatoire avant écriture (CODE_QUALITY_STANDARDS §6) [-99;+99] m
    IF (TargetPositionM < -99.0) OR (TargetPositionM > 99.0) THEN
        TargetOutOfRangeError := TRUE;
    ELSE
        TargetPoints := REAL_TO_DINT(TargetPositionM * UDINT_TO_REAL(PointsPerRev) / CableM_PerRev);
        PendingHomingRefRaw := DINT_TO_UDINT(UDINT_TO_DINT(RawPos) - TargetPoints);
        PresetValue := RawPos;
        PresetRequest := TRUE;
        PresetVerificationActive := TRUE;
        PendingProvisional := ProvisionalHoming;
        Lifecycle.Done := FALSE;
    END_IF;
END_IF;
{endregion}

{region "§5 Suivi de transaction preset"}
// ⏳ 5. SUIVI DE LA TRANSACTION PRESET
PresetVerifyTimer(IN := PresetVerificationActive, PT := CST_PresetVerifyTime);
IF PresetVerificationActive AND PresetVerifyTimer.Q THEN
    CandidateRawDiff := UDINT_TO_DINT(RawPos) - UDINT_TO_DINT(PendingHomingRefRaw);
    IF PointsPerRev <> 0 THEN
        CandidateCablePosM := DINT_TO_REAL(CandidateRawDiff) * CableM_PerRev / UDINT_TO_REAL(PointsPerRev);
    ELSE
        CandidateCablePosM := 0.0;
    END_IF;
    ReadbackOk := ABS(CandidateCablePosM - TargetPositionM) <= CST_HomingVerifyToleranceM;
    StatusBitOk := PresetStatusBit;

    CASE Cfg.PresetConfirmMode OF
        E_PresetConfirmMode.READBACK_ONLY:
            PresetConfirmed := ReadbackOk;
        E_PresetConfirmMode.READBACK_AND_STATUSBIT:
            PresetConfirmed := ReadbackOk AND StatusBitOk;
        E_PresetConfirmMode.STATUSBIT_ONLY:
            PresetConfirmed := StatusBitOk;
        ELSE
            PresetConfirmed := FALSE;
    END_CASE;

    IF PresetConfirmed THEN
        Calib.HomingRefRaw := PendingHomingRefRaw;
        Calib.Homed := TRUE;
        Calib.HomingSuspect := FALSE;
        Calib.HomingProvisional := PendingProvisional;
        Calib.LastKnownRawPos := RawPos;
        PresetConfirmationFailed := FALSE;
        PresetFailError := FALSE;
        Lifecycle.Done := TRUE;
    ELSE
        Calib.HomingSuspect := TRUE;
        Calib.HomingProvisional := FALSE;
        PresetConfirmationFailed := TRUE;
        PresetFailError := TRUE;
        Lifecycle.Done := FALSE;
    END_IF;

    PendingProvisional := FALSE;
    PresetVerificationActive := FALSE;
    PresetVerifyTimer(IN := FALSE, PT := CST_PresetVerifyTime);
END_IF;
{endregion}

{region "§6 Sorties état & calibration"}
// 📤 6. SORTIES ÉTAT & CALIBRATION
IF EncoderAvailable AND NOT PresetVerificationActive THEN
    Calib.LastKnownRawPos := RawPos;
END_IF;

Lifecycle.Busy := PresetVerificationActive;
Homed := Calib.Homed AND NOT Calib.HomingSuspect;
HomingSuspect := Calib.HomingSuspect;
HomingProvisional := Calib.HomingProvisional;
HomingRefRaw := Calib.HomingRefRaw;
{endregion}

          
END_FUNCTION_BLOCK

(* ======================================================================= 🛡️ FB_Encoder_Safety — Bornage physique & surveillance cohérence ─────────────────────────────────────────────────────────────── 🎯 Rôle : Bornage physique absolu [-99; +99]m et relais d'incohérence redémarrage 🔒 Polarité : EncoderIncoherent=TRUE en cas de hors bornes ou HomingSuspect 🛡️ Sécurité : Verrouillage de la position câble sûre 📄 Doc métier : DOC/AF/AF_Partie-09_Fonction_Encoder_v2.4.md ======================================================================= *)
FUNCTION_BLOCK FB_Encoder_Safety
  VAR_INPUT
    Enable : BOOL;  (* === COMMANDES & AUTORISATIONS === --> [CMD] Autorisation generale FB (TRUE=Autorise) *)
    Reset : BOOL;  (* --> [CMD] Acquittement defaut (front montant) *)
    CablePosM : REAL;  (* === MESURES & ALERTE HOMING === --> [HW] Position calculee (m, sortie FB_Encoder_Scale) *)
    HomingSuspect : BOOL;  (* --> [SAFE] Alerte incoherence redemarrage (FB_Encoder_Homing) *)
    PositionMinM : REAL := -99;  (* === REGLAGES & BORNES PHYSIQUES === --> [CFG] Plafond bornage physique bas (m) *)
    PositionMaxM : REAL := 99;  (* --> [CFG] Plafond bornage physique haut (m) *)
    BypassGlobal : BOOL := FALSE;  (* === TESTS & BYPASS === --> [TST] Neutralisation defaut de bornage pour mise en service *)
  END_VAR
  VAR_OUTPUT
    Ready : BOOL;  (* === ETATS IEC & SYNOPTIQUE === <-- [STAT] FB pret a fonctionner *)
    Fault : ST_Fault;  (* 🧩 Statut transverse (forme cible ST_Fault) *)
    CablePosMSafe : REAL;  (* === MESURES SURE & SECURITE === <-- [DIAG] Position cable instantanee transmise (m) *)
    EncoderIncoherent : BOOL;  (* <-- [SAFE] Incoherence ou hors bornes (TRUE = defaut) *)
  END_VAR
  VAR
    ResetEdge : R_TRIG;  (* === DETECTEURS DE FRONT === . [LOC] Detecteur front montant Reset *)
    instFault : FB_FaultCore;  (* === SOCLE DEFAUT (FB_FaultCore) === * [INST] Socle défaut transverse *)
    instCauses : ARRAY[0..15] OF ST_FaultCause;  (* . [LOC] Table des causes nommées *)
  END_VAR

            

// === IMPLEMENTATION ===

{region "§1 Causes & Socle Défaut (évalué en continu)"}
// 🔑 1. RESET FRONT
ResetEdge(CLK := Reset);

// 🔍 2. SURVEILLANCE BORNAGE & INCOHÉRENCE BOOT
instCauses[0].Active   := NOT BypassGlobal AND ((CablePosM < PositionMinM) OR (CablePosM > PositionMaxM));
instCauses[0].Latching := FALSE;
instCauses[0].Texte    := 'Depassement bornes physiques absolues cable';

instCauses[1].Active   := NOT BypassGlobal AND HomingSuspect;
instCauses[1].Latching := FALSE;
instCauses[1].Texte    := 'Incoherence position au redemarrage';

// Appel du socle de défaut
instFault(Enable := Enable, Reset := Reset, Causes := instCauses);
Fault := instFault.Fault;
{endregion}

{region "§2 Gate neutralisation"}
// 🛑 2. GATE
IF NOT Enable THEN
    Ready := FALSE;
    CablePosMSafe := CablePosM;
    EncoderIncoherent := FALSE;
    RETURN;
END_IF;

Ready := Enable AND NOT Fault.Latched;
{endregion}

{region "§3 Transmission mesure et sécurité"}
// 📏 3. TRANSMISSION DE LA MESURE & SÉCURITÉ
CablePosMSafe := CablePosM;
EncoderIncoherent := Fault.Error;
{endregion}

          
END_FUNCTION_BLOCK

(* ======================================================================= ⚙️ FB_Encoder_Scale — Mise à l'échelle points → mètres (1 par treuil) ─────────────────────────────────────────────────────────────── 🎯 Rôle : Calcul de la position câble en mètres par conversion arithmétique signée 🔒 Polarité : CablePosM signée (+ enroulé, - sous l'eau) 🔌 Architecture : Convertisseur de mesure unitaire par treuil 📄 Doc métier : DOC/AF/AF_Partie-09_Fonction_Encoder_v2.4.md ======================================================================= === DECLARATION (à coller dans la partie déclaration du POU FB_Encoder_Scale) === *)
FUNCTION_BLOCK FB_Encoder_Scale
  VAR_INPUT
    RawPos : UDINT;  (* === DONNEES ENTREE & REFERENCES BRUTES === --> [HW] Position brute codeur (sortie FB_Encoder_Abs, gelee sur doute) *)
    HomingRefRaw : UDINT;  (* --> [CFG] Reference brute figee au dernier homing (ST_Encoder_Calib) *)
    CableM_PerRev : REAL := 2;  (* === PARAMETRES & RATIOS DE CONVERSION === --> [CFG] Developpement cable par tour tambour (m/tour) *)
    PointsPerRev : UDINT := 8192;  (* --> [CFG] Resolution codeur (pts/tour) *)
  END_VAR
  VAR_OUTPUT
    CablePosM : REAL;  (* === MESURE CONVERTIE === <-- [DIAG] Position cable en metres (+ enroule, - sous l'eau) *)
  END_VAR
  VAR
    RawDiff : DINT;  (* === CALCULS INTERNES === . [LOC] Ecart signe RawPos - HomingRefRaw *)
  END_VAR

            

// === IMPLEMENTATION (à coller dans le corps ST du POU FB_Encoder_Scale) ===

// 🧮 Écart signé sûr : conversion DINT AVANT soustraction (§3.1) — jamais l'inverse
RawDiff := UDINT_TO_DINT(RawPos) - UDINT_TO_DINT(HomingRefRaw);

// 📏 Formule fixe points → mètres (Partie10 §2), garde division par zéro
IF PointsPerRev > 0 THEN
    CablePosM := DINT_TO_REAL(RawDiff) * (CableM_PerRev / UDINT_TO_REAL(PointsPerRev));
ELSE
    CablePosM := 0.0;
END_IF;

          
END_FUNCTION_BLOCK

(* ======================================================================= ⚙️ FB_Encoder_SpeedMeasure — Mesure de vitesse câble directe codeur ─────────────────────────────────────────────────────────────── 🎯 Rôle : Conversion directe du mot de vitesse natif codeur EtherCAT (m/s) ⚙️ Source CoE : Objet 0x6031:01 en 0.1 RPM (dixième de tour/min) 📐 Formule : V(m/s) = (SpdValue * 0.1 * CableM_PerRev) / 60.0 🛡️ Sans bornage : zéro clamping artificiel, suppression délai filtre PT1 📄 Doc métier : DOC/AF/AF_Partie-09_Fonction_Encoder_v2.4.md ======================================================================= *)
FUNCTION_BLOCK FB_Encoder_SpeedMeasure
  VAR_INPUT
    Enable : BOOL;  (* === COMMANDES & AUTORISATIONS === --> [CMD] Autorisation generale FB (TRUE=Autorise) *)
    Reset : BOOL;  (* --> [CMD] Purge immediate (front montant) *)
    SpdValueIn : DINT;  (* === MESURES EN ENTREE === --> [HW] Mot de vitesse brut EtherCAT (0x6031:01 en 0.1 RPM) *)
    PositionValid : BOOL;  (* --> [SAFE] Validite de la chaine codeur *)
    CableM_PerRev : REAL := 2;  (* --> [CFG] Developpement cable par tour tambour (m/tour) *)
  END_VAR
  VAR_OUTPUT
    Speed_Mps : REAL;  (* === VITESSE CÂBLE QUALIFIÉE (m/s) === <-- [DIAG] Vitesse absolue directe (m/s) *)
    SignedSpeed_Mps : REAL;  (* <-- [DIAG] Vitesse signee directe (+ montee, - descente) (m/s) *)
    Valid : BOOL;  (* <-- [STAT] Validite mesure (TRUE si codeur operationnel et autorise) *)
  END_VAR
  VAR
    ResetEdge : R_TRIG;  (* === MEMOIRES & DETECTEURS === . [LOC] Detecteur front montant Reset *)
  END_VAR

            

{region "§1 Gate de neutralisation & Reset"}
ResetEdge(CLK := Reset);

// Purge immediate sur perte de confiance, desactivation ou Reset
IF NOT Enable OR ResetEdge.Q OR NOT PositionValid THEN
    Speed_Mps       := 0.0;
    SignedSpeed_Mps := 0.0;
    Valid           := FALSE;
    RETURN;
END_IF;
{endregion}

{region "§2 Conversion directe vitesse CoE (0.1 RPM -> m/s)"}
// Formule cinematique directe :
// N_RPM = SpdValueIn * 0.1
// V_mps = (N_RPM * CableM_PerRev) / 60.0 = (DINT_TO_REAL(SpdValueIn) * 0.1 * CableM_PerRev) / 60.0
SignedSpeed_Mps := (DINT_TO_REAL(SpdValueIn) * 0.1 * CableM_PerRev) / 60.0;
Speed_Mps       := ABS(SignedSpeed_Mps);
Valid           := TRUE;
{endregion}

          
END_FUNCTION_BLOCK

(* ======================================================================= 🧩 FB_FaultCore — Socle de remplissage de ST_Fault (vue live + vue latchée) ─────────────────────────────────────────────────────────────── 🎯 Rôle : à partir d'une LISTE de causes en clair (ARRAY[0..15] OF ST_FaultCause), produire la brique ST_Fault : • Error / ErrorId : vue LIVE, suit les causes Active, retombe seule. • Latched / LatchedId: vue LATCHÉE, chaque bit figé à l'apparition d'une cause `Active AND Latching`, conservé jusqu'au front Reset. 🔒 Sécurité : - interlock TOUJOURS sur `Causes[i].Active` (cause brute), jamais sur le latch. - Reset TOUJOURS effectif, jamais conditionné (std §9) — agit même Enable=FALSE. - Latching=FALSE → cause visible en LIVE seulement (fail-safe : reste visible). - un défaut laté non acquitté reste publié même FB désactivé (pas d'effacement silencieux sur bascule Enable OFF→ON sans Reset). - une cause à acquitter réapparue re-arme son bit (ré-alarme). 🧬 Un seul socle, réutilisé par tout FB `standard` qui expose un ST_Fault. Pas de State, pas de Warning, pas de texte — hors périmètre de ce socle. 📄 Doc : DOC/STDS/CODE_QUALITY_STANDARDS.md §2quinquies / §9 ======================================================================= *)
FUNCTION_BLOCK FB_FaultCore
  VAR_INPUT
    Enable : BOOL;  (* --> [CMD] Autorisation générale du FB porteur *)
    Reset : BOOL;  (* --> [CMD] Front d'acquittement (jamais conditionné, §9) *)
    Causes : ARRAY[0..15] OF ST_FaultCause;  (* --> [CMD] Liste des causes en clair (Active / Latching / Texte) *)
  END_VAR
  VAR_OUTPUT
    Ready : BOOL;  (* <-- [STAT] FB porteur autorisé (= Enable) *)
    Fault : ST_Fault;  (* <-- [DIAG] Brique défaut (mappée 1:1 sur la sortie du FB porteur) *)
  END_VAR
  VAR
    ResetEdge : R_TRIG;  (* . [LOC] Front montant Reset *)
    Latch : ARRAY[0..15] OF BOOL;  (* . [LOC] Bit laté par cause, jusqu'au Reset *)
    i : INT;  (* . [LOC] Index de parcours de la liste *)
  END_VAR

            

{region "§1 Reset (front, toujours effectif)"}
// Front Reset : efface tous les latches. Jamais conditionné, agit même Enable=FALSE (§9).
Ready := Enable;
ResetEdge(CLK := Reset);
IF ResetEdge.Q THEN
    FOR i := 0 TO 15 DO Latch[i] := FALSE; END_FOR;
END_IF;
{endregion}

{region "§2 Vue LIVE — Error / ErrorId"}
// Bitfield des causes présentes MAINTENANT. Retombe seule à 0 quand les causes disparaissent.
// Non évaluée si Enable=FALSE (pas de lecture de cause hors autorisation).
Fault.ErrorId := 0;
IF Enable THEN
    FOR i := 0 TO 15 DO
        IF Causes[i].Active THEN
            Fault.ErrorId := Fault.ErrorId OR SHL(WORD#1, INT_TO_DWORD(i));
        END_IF;
    END_FOR;
END_IF;
Fault.Error := (Fault.ErrorId <> 0);
{endregion}

{region "§3 Armement des latches (causes à acquitter)"}
// Une cause Active ET Latching arme son bit ; le bit reste jusqu'au front Reset (§1),
// même si la cause disparaît. Réapparition => ré-armement (ré-alarme).
IF Enable THEN
    FOR i := 0 TO 15 DO
        IF Causes[i].Active AND Causes[i].Latching THEN
            Latch[i] := TRUE;
        END_IF;
    END_FOR;
END_IF;
{endregion}

{region "§4 Vue LATCHÉE — Latched / LatchedId"}
// Toujours publiée, y compris Enable=FALSE : un défaut non acquitté reste visible.
Fault.LatchedId := 0;
FOR i := 0 TO 15 DO
    IF Latch[i] THEN
        Fault.LatchedId := Fault.LatchedId OR SHL(WORD#1, INT_TO_DWORD(i));
    END_IF;
END_FOR;
Fault.Latched := (Fault.LatchedId <> 0);
{endregion}

          
END_FUNCTION_BLOCK
